// TwinCAT 3 PLC project ExternControl
// ProgramVersion: 3.1.4026.19
// libraries:
//   Tc2_Standard, * (Beckhoff Automation GmbH)
//   Tc2_System, * (Beckhoff Automation GmbH)
//   Tc2_Utilities, * (Beckhoff Automation GmbH)
// project tree:
//   / GlobalTextList.TcGTLO (not stored), MAIN.TcPOU, PlcTask.TcTTO, Visualization Manager.TcVMO (not stored)
//   MAPPING/ MAPPING_out.TcPOU, MAPPING_in.TcPOU
//   MAPPING/types/ U_AXIS_CTRL.TcDUT, U_AXIS_GEAR_IN.TcDUT, U_AXIS_HOMING.TcDUT (not stored), U_AXIS_INFO.TcDUT (not stored), U_AXIS_MOTION_OPTIONS.TcDUT (not stored), U_AXIS_MOVE_DATA.TcDUT (not stored), U_AXIS_NC_PARAMETER_RD.TcDUT (not stored), U_AXIS_NC_PARAMETER_WRT.TcDUT, U_AXIS_STATE.TcDUT (not stored)
//   NC_PTP/types/axis/ E_AxisEncoderType.TcDUT (not stored), ST_HomeParams.TcDUT, ST_HomingOptionsExt.TcDUT (not stored)
//   NC_PTP/types/control/ E_AXIS_CTRL.TcDUT (not stored), E_AXIS_STATE.TcDUT (not stored), ST_AXIS_CTRL.TcDUT (not stored), ST_AXIS_INFO.TcDUT, ST_AXIS_STATE.TcDUT (not stored), ST_GEAR_IN.TcDUT (not stored), ST_HOMING.TcDUT (not stored), ST_MOTION_OPTIONS.TcDUT (not stored), ST_MOVE_DATA.TcDUT, ST_NC_PARAMETER.TcDUT (not stored)
//   _GVL/ GVL_AXIS.TcGVL (not stored), GVL_MSG.TcGVL, PLC_CONSTANT.TcGVL (not stored)
//   _DUT/ E_CHECK_STATE.TcDUT (not stored), E_PROGRESS.TcDUT (not stored)
//   _MSG/ fb_LocalTime.TcPOU (not stored), f_MessageSet.TcPOU (not stored), MessageData.TcPOU (not stored), T_MESSAGE_LIST.TcVIS (not stored)
//   _MSG/types/ e_Device.TcDUT, E_MessageType.TcDUT, E_MESSAGE_STATE.TcDUT, e_Subdevice.TcDUT, ST_Message.TcDUT (not stored)
// (motion and I/O tree: see PLC project plc_motion)
// real-time tasks:
//   TASK PlcTask: cycle T#10ms, priority 20, ADS port 350
//   TASK PlcTask1: cycle T#10ms, priority 21, ADS port 351
// variable links:

CONFIGURATION ExternControl
    RESOURCE PLC ON TwinCAT3
        TASK PlcTask(INTERVAL := T#10ms, PRIORITY := 21);
        PROGRAM MAPPING_in WITH PlcTask : MAPPING_in;
        PROGRAM MAIN WITH PlcTask : MAIN;
        PROGRAM MAPPING_out WITH PlcTask : MAPPING_out;
    END_RESOURCE
END_CONFIGURATION

// ---- MAPPING/types/U_AXIS_CTRL.TcDUT
TYPE U_AXIS_CTRL :
UNION

  stCtrl              : ARRAY[1..MAX_AXIS] OF ST_AXIS_CTRL;

  byCtrl    AT %Q*    : ARRAY[1..MAX_AXIS] OF
                        ARRAY[1..SIZEOF(ST_AXIS_CTRL)] OF BYTE;
END_UNION
END_TYPE

// ---- MAPPING/types/U_AXIS_GEAR_IN.TcDUT
TYPE U_AXIS_GEAR_IN :
UNION

  stCtrl              : ARRAY[1..MAX_AXIS] OF ST_GEAR_IN;

  byCtrl    AT %Q*    : ARRAY[1..MAX_AXIS] OF
                        ARRAY[1..SIZEOF(ST_GEAR_IN)] OF BYTE;
END_UNION
END_TYPE

// ---- MAPPING/types/U_AXIS_NC_PARAMETER_WRT.TcDUT
TYPE U_AXIS_NC_PARAMETER_WRT :
UNION

  stCtrl              : ARRAY[1..MAX_AXIS] OF ST_NC_PARAMETER;

  byCtrl    AT %Q*    : ARRAY[1..MAX_AXIS] OF
                        ARRAY[1..SIZEOF(ST_NC_PARAMETER)] OF BYTE;
END_UNION
END_TYPE

// ---- NC_PTP/types/axis/ST_HomeParams.TcDUT
TYPE ST_HomeParams :
STRUCT
  Position              : LREAL;
  HomingMode            : INT;
  Options               : ST_HomingOptionsExt;

  InvertHomeSensor      : BIT := FALSE;   //Set to true,  NormallyClosed home sensor
  SimulateHomeSensor    : BIT := FALSE;   //Set to true,  homed on encoder index only. The homing methode 'hardware sync' must be used then.

  UseLimitMin           : BIT := TRUE;    //Set to false, no negative limit sensor.

  InvertLimitMin        : BIT := FALSE;   //Set to true,  NC negative limit sensor
  HomeOnLimitMin        : BIT := FALSE;   //Set to true,  homed on negative limit sensor 

  UseLimitMax           : BIT := TRUE;    //Set to false, no positive limit sensor.

  InvertLimitMax        : BIT := FALSE;   //Set to true,  NC positive limit sensor
  HomeOnLimitMax        : BIT := FALSE;   //Set to true,  homed on positive limit sensor 
  
  // It is not allowed to use more than 1 of the 3 switches: SimulateHomeSensor, HomeOnLimitMin, HomeOnLimitMax
  
END_STRUCT
END_TYPE

// ---- NC_PTP/types/control/ST_AXIS_INFO.TcDUT
{attribute 'pack_mode' := '2'}
TYPE ST_AXIS_INFO :
STRUCT
  bEnabled    : BIT; // Enabled: check if ControlLoop is closed and active
  bReferenced : BIT; // Axis homing bit
  bReady      : BIT; // enabled & NOT bError & no Axis Function requested
  bBusy       : BIT; // axis function requested or active
  bError      : BIT;
  bTimeout    : BIT; // for move cmds or switching drive on timeout
  bInTarget   : BIT; // ActPos = SetPos --> position check is done with configured window in NC
  bStandstill : BIT; // No Error and NOT moving
 
  nErrorId            : UDINT;

  rActPos             : LREAL;
  rActVelo            : LREAL;
  rPosDiff            : LREAL;

  dwCoupleState       : DWORD;   // cyclic information about axis couple state
  nNcAxisId           : UDINT;
END_STRUCT
END_TYPE

// ---- NC_PTP/types/control/ST_MOVE_DATA.TcDUT
{attribute 'pack_mode' := '2'}
TYPE ST_MOVE_DATA :
STRUCT
  rSetPos           : LREAL;
  rSetVelo          : LREAL;
  rOverride         : LREAL := 100.0;
  rAcc              : LREAL;
  rDec              : LREAL;
  rJerk             : LREAL;
  iDirection        : INT;
END_STRUCT
END_TYPE

// ---- _MSG/types/e_Device.TcDUT
{attribute 'to_string'}
TYPE e_Device :
(
  Device_Null,
  General           :=  1000,
  CaGroup           :=  2000,
  Xpu               :=  3000,
  XpuCtrl           :=  4000,
  Mover             :=  5000,
  MoverCtrl         :=  6000,
  XtsTransportUnit  :=  7000,
  XfcTriggerBox     :=  8000,
  XfcTouchProbe     :=  9000,
  XtsStation        := 10000,

  Camming           := 11000,
  NciChannel        := 12000,
  NciChannelCtrl    := 13000,
  Axis              := 14000,
  XfcAxis           := 15000,
  Data              := 16000,

  Process           := 20000,
  Application       := 30000
)UDINT;
END_TYPE

// ---- _MSG/types/E_MessageType.TcDUT
{attribute 'strict'}
{attribute 'to_string'}
TYPE E_MessageType :
(
  eMessageEmpty,
  eMessageError,
  eMessageWarning,
  eMessageInfo,
  eMessageVerbose
)DINT;
END_TYPE

// ---- _MSG/types/E_MESSAGE_STATE.TcDUT
{attribute 'strict'}
TYPE E_MESSAGE_STATE :
(
  MSG_INVALID_POINTERS  := -1,
	MSG_NULL,
  MSG_INIT,
  MSG_ROOT              := 10,
  MSG_ROOT_CREATE,
  MSG_ROOT_CREATE_BUSY,
  MSG_FOLDER,
  MSG_FOLDER_CREATE,
  MSG_FOLDER_CREATE_BUSY,
  MSG_FILE_CREATE_DONE,
  MSG_LINE_START        := 100,
  MSG_LINE_BUILD,
  MSG_LINE_CHECK,
  MSG_WRITE_FILE_BUSY  := 200,
  MSG_WRITE_FILE_END,
  MSG_WRITE_FILE_DONE   := 1000
)DINT;
END_TYPE

// ---- _MSG/types/e_Subdevice.TcDUT
{attribute 'strict'}
{attribute 'to_string'}
TYPE e_Subdevice :
(
  // sub device for message system
  General                 :=  0,
  // Motion Control
  fbPower,
  fbReset,
  fbResetSercos,
  fbHalt,
  fbStop,                 // 5
  fbHome,
  fbJog,
  fbMoveVelocity1,
  fbMoveVelocity2,
  fbMoveAbsolute1,        // 10
  fbMoveAbsolute2,
  fbMoveEndless,
  fbMovePtP,
  fbMoveVelo,
  fbSendToPos,

  // CA CollisionAvoidance FB instances
  // CA group fb instances
  fbCaGroup             := 30,
  fbMoveToPosCa,
  fbSendToAbsPosCa,
  fbSendToModuloPosCa,
  fbGearInPosCa,
  fbGroupAddAxis,
  fbGroupRemoveAxis,
  fbGroupDisable,
  fbGroupEnable,
  fbGroupErrorRead,
  fbGroupStatusRead,
  fbGroupReset,
  fbGroupStop,

  fbGearIn              := 50,
  fbGearOut,
  fbGearInMultiMaster,

  fbCamOut              := 80,
  fbCamInV2,
  fbCamScalingV2,
  fbCamInfoV2,
  fbReadMotionFunction,
  fbReadMotionFunctionPoint,
  fbReadMotionFunctionValues,
  fbWriteMotionFunction,
  fbWriteMotionFunctionPoint,
  fbSetOnlineChangeMode,

  fbReadParameter       := 100,
  fbReadBoolParameter,
  fbWriteParameter,
  fbWriteBoolParameter,
  fbWriteParameterPersistent,

	fbBuildGroup          := 200,
	fbClearGroup,
	fbLoadProg,
	fbResetItp,
	fbStartStopItp,
	fbEStopItp,
	fbStepOnAfterEStopItp,
	fbConfirmHskItp,
	fbDelDtgItp,
	fbNciFeedTablePreparation,
	fbNciFeedTable,
	fbReadLine,
  fbItpReadRParams,
  fbItpWriteRParams,
  Get_ItpState,
  Get_Error,

  XfcPositionAtTime       := 300,
  XfcTimeOfPosition,
  XfcTimeToPosition,
  XfcTimeToModuloPosition,
  XfcRecordedPosition,
  XfcTouchProbe,          // 305
  XfcTouchProbeEL1258,
  XfcTouchProbeOptions,
  XfcTriggerRef,
  XfcTriggerRef_MT,
  XfcEl1258Interface_MT,  // 310
  XfcRecordedPosition_MT,
  XfcTriggerOut,
  XfcTriggerStart,
  XfcSwitchOn_2252,
  XfcSwitchOff_2252,      // 315
  XfcInit,
  XfcLatchPosition,
  XfcWaitForPosition,

  AxisControl           := 1000,
  AxisStartUp,
  AxisCycle,
  AxisIdle,

  NciControl           := 2000,
  NciStartUp,
  NciCycle,
  NciIdle,

  StationLinkedList     := 3000,
  StationInitList,
  StationAddHead,
  StationAddTail,
  StationGetHead,
  StationRemoveHeadValue,

  StationControl        := 4000,
  StationState, 

  Xpu_fbEnvironment     := 5000,
  Xpu_fbProcessingUnit,
  Xpu_fbXpuPart,
  Xpu_fbXpuTrack,
  Xpu_fbMc2CaGroup,
  Xpu_fbParameterSet,
  Xpu_fbNctController,

  Xpu_fbPartModules     := 5500,

  Xpu_fbMoverXpu        := 6000,

  Xpu_fbNctBaseUnit     := 6500,

  TransportUnit_General := 7000,
  TransportUnit_Restart := 7010,
  TransportUnit_Start,
  TransportUnit_XpuInit,
  TransportUnit_StationClearOutfeed,

  CamControl            := 8000,
  CamStartUp,
  CamCycle,

  Process_StationCollector    := 11000,
  Process_Process_Collector   := 11100,
  Process_ProcessCollector_Init,
  Process_ProcessCollector_Cycle,
  Process_ProcessCollector_Control,

  Process_LinkedList_GetHead,
  Process_LinkedList_RemoveHead,
  Process_LinkedList_AddTail

)uDINT;
END_TYPE

// ---- _GVL/GVL_MSG.TcGVL
{attribute 'qualified_only'}
VAR_GLOBAL CONSTANT
  //-----------------------------------------------------------------------------
  // file paths for message system
  //  - compiler define option WIN switches to Windows file paths
  //-----------------------------------------------------------------------------
{IF NOT defined (BSD)}
  {info 'PLC_MOTION_LAYER: WIN'}
  LOG_DIR               : STRING  := 'C:\TwinCAT\#MsgFiles\';
{ELSE}
  {info 'PLC_MOTION_LAYER: BSD'}
  LOG_DIR               : STRING  := '/usr/local/etc/TwinCAT/#MsgFiles/';
{END_IF}

  LOG_FILE              : STRING  := 'MSG_EXT_';

  MAX_MESSAGE           : UINT     := 200; // max entry in message list
END_VAR
VAR_GLOBAL
  fbLocalTime                     : fb_LocalTime;
  dtLocalTime                     : DT;
  sLocalTime                      : STRING;

  Messages                        : ARRAY[1..MAX_MESSAGE] OF ST_Message;
  MessageIndex                    : UINT := 0; // message index
  MessageError                    : UINT := 0; // error counter

  MessageLevelAxisPtp             : E_MessageType := E_MessageType.eMessageError;
  MessageLevelAxisCam             : E_MessageType := E_MessageType.eMessageError;
  MessageLevelNciChn              : E_MessageType := E_MessageType.eMessageError;

  MessageLevelTriggerBox          : ARRAY[1..PLC_CONSTANT.MAX_TRIGGER_BOX]  OF E_MessageType;
  MessageLevelTouchProbe          : ARRAY[1..PLC_CONSTANT.MAX_TOUCH_PROBE]  OF E_MessageType;


  // diag data
  dbg_AxisIdxGearIn               : ARRAY[1..PLC_CONSTANT.MAX_AXIS]      OF BYTE; // diag for Axis gear in
  dbg_AxisIdxGearInMultiMaster    : ARRAY[1..PLC_CONSTANT.MAX_AXIS,1..4] OF BYTE; // diag for Axis gear in multi master
  dbg_AxisIdxCamIn                : ARRAY[1..PLC_CONSTANT.MAX_AXIS]      OF BYTE; // diag for Axis cam in
END_VAR

// ---- MAPPING/MAPPING_in.TcPOU
PROGRAM MAPPING_in
VAR
  bFirstCycle       : BOOL := TRUE;

  AxisState         : U_AXIS_STATE;
  AxisInfo          : U_AXIS_INFO;
  AxisParameterRd   : U_AXIS_NC_PARAMETER_RD;

  szAxisPara,
  szAxisInfo,
  szAxisState           : ARRAY[1..2] OF UDINT;

  szCamInfo,
  szCamData,
  szCamState            : ARRAY[1..2] OF UDINT;

  szStateTouchProbe,
  szStateTrigger	      :  ARRAY[1..2] OF UDINT;
END_VAR


IF (bFirstCycle)
THEN
  bFirstCycle         := FALSE;
  
  szAxisState[1]      := SIZEOF(AxisState);
  szAxisState[2]      := SIZEOF(GVL_AXIS.State);
  
  szAxisInfo [1]      := SIZEOF(AxisInfo);
  szAxisInfo [2]      := SIZEOF(GVL_AXIS.Info);
  
  szAxisPara [1]      := SIZEOF(AxisParameterRd);
  szAxisPara [2]      := SIZEOF(GVL_AXIS.NcParameterRd);
END_IF

  memcpy(ADR(GVL_AXIS.State),         ADR(AxisState),              SIZEOF(AxisState));
  memcpy(ADR(GVL_AXIS.Info),          ADR(AxisInfo),               SIZEOF(AxisInfo));
  memcpy(ADR(GVL_AXIS.NcParameterRd), ADR(AxisParameterRd),        SIZEOF(AxisParameterRd));

END_PROGRAM

// ---- MAIN.TcPOU
PROGRAM MAIN
VAR
  nAxis     : UINT;

END_VAR




//-----------------------------------------------------------------------------------------------------------------
//-----------------------------------------------------------------------------------------------------------------
// react to operation modes (how to do it in an easy self documenting way)
//-----------------------------------------------------------------------------------------------------------------
//-----------------------------------------------------------------------------------------------------------------
CASE (GVL_AXIS.State[nAxis].eState MOD E_PROGRESS.PROGRESS_DONE)
OF
  E_AXIS_STATE.AXIS_INIT:
    ;// do something after success  

  E_AXIS_STATE.AXIS_MOVE_POS:
    ;// do something after success
ELSE
  CASE (GVL_AXIS.State[nAxis].eState MOD E_PROGRESS.PROGRESS_ERROR)
  OF
    E_AXIS_STATE.AXIS_INIT:
      ;// do something after success  
  
    E_AXIS_STATE.AXIS_MOVE_POS:
      ;// do something after success
  ELSE
    ;// down the rabbit hole you go from here
  END_CASE
END_CASE

END_PROGRAM

// ---- MAPPING/MAPPING_out.TcPOU
PROGRAM MAPPING_out
VAR
  bFirstCycle       : BOOL := TRUE;

  AxisCtrl          : U_AXIS_CTRL;
  AxisMoveData      : U_AXIS_MOVE_DATA;
  AxisMotionOptions : U_AXIS_MOTION_OPTIONS;

  AxisGearInData    : U_AXIS_GEAR_IN;
  AxisHoming        : U_AXIS_HOMING;
  AxisParameterWrt  : U_AXIS_NC_PARAMETER_WRT;

  szAxisPara,
  szAxisHoming,
  szAxisGearData,
  szAxisMotionOptions,
  szAxisMoveData,
  szAxisCtrl          : ARRAY[1..2] OF UDINT;

  szCamCtrl           : ARRAY[1..2] OF UDINT;

  szCtrlTouchProbe,
  szCtrlTrigger       :  ARRAY[1..2] OF UDINT;
END_VAR


IF (bFirstCycle)
THEN
  bFirstCycle             := FALSE;

  szAxisCtrl[1]           := SIZEOF(AxisCtrl);
  szAxisCtrl[2]           := SIZEOF(GVL_AXIS.Ctrl);
  
  szAxisMoveData [1]      := SIZEOF(AxisMoveData);
  szAxisMoveData [2]      := SIZEOF(GVL_AXIS.Data);
  
  szAxisMotionOptions [1] := SIZEOF(AxisMotionOptions);
  szAxisMotionOptions [2] := SIZEOF(GVL_AXIS.MotionOptions);
  
  szAxisGearData [1]      := SIZEOF(AxisGearInData);
  szAxisGearData [2]      := SIZEOF(GVL_AXIS.GearInParameter);
  
  szAxisHoming [1]        := SIZEOF(AxisHoming);
  szAxisHoming [2]        := SIZEOF(GVL_AXIS.HomeParameter);
  
  szAxisPara [1]          := SIZEOF(AxisParameterWrt);
  szAxisPara [2]          := SIZEOF(GVL_AXIS.NcParameterWrt);
  
END_IF

  memcpy(ADR(AxisCtrl),                 ADR(GVL_AXIS.Ctrl),             SIZEOF(AxisCTrl));
  memcpy(ADR(AxisMoveData),             ADR(GVL_AXIS.Data),             SIZEOF(AxisMoveData));
  memcpy(ADR(AxisMotionOptions),        ADR(GVL_AXIS.MotionOptions),    SIZEOF(AxisMotionOptions));
  
  memcpy(ADR(AxisGearInData),           ADR(GVL_AXIS.GearInParameter),  SIZEOF(AxisGearInData));
  memcpy(ADR(AxisHoming),               ADR(GVL_AXIS.HomeParameter),    SIZEOF(AxisHoming));
  memcpy(ADR(AxisParameterWrt),         ADR(GVL_AXIS.NcParameterWrt),   SIZEOF(AxisParameterWrt));

END_PROGRAM
